// SIMATIC STEP 7 (V5.x) project Mikser
// CPU: CPU 317-2 PN/DP
// station: Hardware
// station: SIMATIC 300(1)
// station: P_ADR_BUS
// program: S7 Program(1)

SYMBOL_TABLE
"CTRL_MIXER"	FC 1	FC 1	// control of simple mixing station
"P1"	I 1.0	BOOL	// wykonaj cykl pracy mieszad³a
"S1"	I 1.1	BOOL	// górny poziom mieszanki w zbiorniku mieszad³a
"S2"	I 1.2	BOOL	// dolny poziom mieszanki w zbiorniku mieszad³a
"Y1"	Q 1.0	BOOL	// sterowanie zaworem dolotowym Y1
"Y2"	Q 1.1	BOOL	// sterowanie zaworem dolotowym Y2
"Y3"	Q 1.2	BOOL	// sterowanie zaworem wylotowym Y3
"K1"	Q 1.3	BOOL	// sterowanie silnikiem mieszad³a
END_SYMBOL_TABLE

FUNCTION "CTRL_MIXER" : VOID	// FC 1
TITLE = CTRL_MIXER
//funkcja steruj¹ca stacj¹ mieszaj¹c¹
//
//                MixerMotor
// In1Valve          ___        In2Valve
//  _|\/|________   | M |   _____|\/|_
//   |/\|        |  |___|  |     |/\|
//               |    |    |
//            |  |    |    |  |_LevelHi
//            |       |       | 
//            |       |       |
//            |      ---      |_LevelLo 
//            |_______________|
//                    |
//                    |  Out1Valve
//                    |____|\/|_  
//                         |/\|
//
VERSION : 0.1
VAR_INPUT
  CycleOn : BOOL ;	//wykonaj pojedynczy cykl: stan aktywny "1"
  LevelLo : BOOL ;	//dolny czujnik poziomu: stan aktywnu "1"
  LevelHi : BOOL ;	//górny czujnik poziomu: stan aktywny "1"
  MixingTime : S5TIME ;	//czas mieszania
  Timer1 : TIMER ;	//timer odliczaj¹cy dzia³anie mieszad³a
END_VAR
VAR_OUTPUT
  In1Valve : BOOL ;	//sterowanie zaworem wlotowym: zamkniêty "0"
  In2Valve : BOOL ;	//sterowanie zaworem wlotowym: zamkniêty "0"
  Out1Valve : BOOL ;	//sterowanie zaworem wylotowym: zamkniêty "1"
  MixerMotor : BOOL ;	//sterowanie silnikiem mieszad³a
END_VAR
VAR_IN_OUT
  CycleMem : BOOL ;	//pamiêæ rozpoczêtego cyklu
END_VAR
VAR_TEMP
  TempBool : BOOL ;
END_VAR
BEGIN
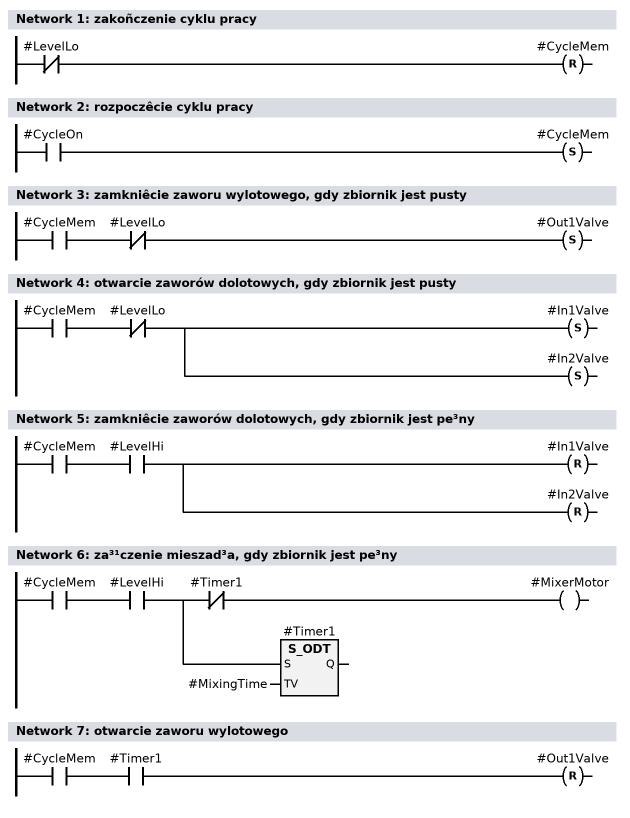
NETWORK
TITLE = zakoñczenie cyklu pracy
      AN    #LevelLo;
      R     #CycleMem;
NETWORK
TITLE = rozpoczêcie cyklu pracy
      A     #CycleOn;
      S     #CycleMem;
NETWORK
TITLE = zamkniêcie zaworu wylotowego, gdy zbiornik jest pusty
      A     #CycleMem;
      AN    #LevelLo;
      S     #Out1Valve;
NETWORK
TITLE = otwarcie zaworów dolotowych, gdy zbiornik jest pusty
      A     #CycleMem;
      AN    #LevelLo;
      S     #In1Valve;
      S     #In2Valve;
NETWORK
TITLE = zamkniêcie zaworów dolotowych, gdy zbiornik jest pe³ny
      A     #CycleMem;
      A     #LevelHi;
      R     #In1Valve;
      R     #In2Valve;
NETWORK
TITLE = za³¹czenie mieszad³a, gdy zbiornik jest pe³ny
//oraz wy³¹czenie mieszad³a po okreœlonym czasie
      A     #CycleMem;
      A     #LevelHi;
      =     L 1.0;
      A     L 1.0;
      AN    #Timer1;
      =     #MixerMotor;
      A     L 1.0;
      L     #MixingTime;
      SD    #Timer1;
      NOP   0;
      NOP   0;
      NOP   0;
      NOP   0;
NETWORK
TITLE = otwarcie zaworu wylotowego
      A     #CycleMem;
      A     #Timer1;
      R     #Out1Valve;
END_FUNCTION

ORGANIZATION_BLOCK OB 1
TITLE = "Main Program Sweep (Cycle)"
VERSION : 0.1
VAR_TEMP
  OB1_EV_CLASS : BYTE ;	//Bits 0-3 = 1 (Coming event), Bits 4-7 = 1 (Event class 1)
  OB1_SCAN_1 : BYTE ;	//1 (Cold restart scan 1 of OB 1), 3 (Scan 2-n of OB 1)
  OB1_PRIORITY : BYTE ;	//Priority of OB Execution
  OB1_OB_NUMBR : BYTE ;	//1 (Organization block 1, OB1)
  OB1_RESERVED_1 : BYTE ;	//Reserved for system
  OB1_RESERVED_2 : BYTE ;	//Reserved for system
  OB1_PREV_CYCLE : INT ;	//Cycle time of previous OB1 scan (milliseconds)
  OB1_MIN_CYCLE : INT ;	//Minimum cycle time of OB1 (milliseconds)
  OB1_MAX_CYCLE : INT ;	//Maximum cycle time of OB1 (milliseconds)
  OB1_DATE_TIME : DATE_AND_TIME ;	//Date and time OB1 started
END_VAR
BEGIN
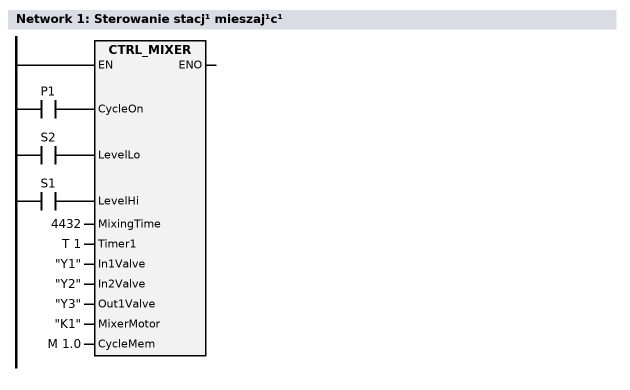
NETWORK
TITLE = Sterowanie stacj¹ mieszaj¹c¹
      A     "P1";
      =     L 20.0;
      BLD   103;
      A     "S2";
      =     L 20.1;
      BLD   103;
      A     "S1";
      =     L 20.2;
      BLD   103;
      CALL  "CTRL_MIXER" (
           CycleOn                  := L 20.0,
           LevelLo                  := L 20.1,
           LevelHi                  := L 20.2,
           MixingTime               := 4432,
           Timer1                   := T 1,
           In1Valve                 := "Y1",
           In2Valve                 := "Y2",
           Out1Valve                := "Y3",
           MixerMotor               := "K1",
           CycleMem                 := M 1.0);
      NOP   0;
END_ORGANIZATION_BLOCK
